// TwinCAT 3 PLC project Intersection
// ProgramVersion: 3.1.4022.2
// libraries:
//   Tc2_Math, * (Beckhoff Automation GmbH)
//   Tc2_Standard, * (Beckhoff Automation GmbH)
//   Tc2_System, * (Beckhoff Automation GmbH)
//   Tc3_Module, * (Beckhoff Automation GmbH)
//   VisuDialogs, * (System)
//   VisuSymbols,3.5.10.0,System
// project tree:
//   01_NorthLight/ NorthLight_Control.TcPOU
//   02_SouthLight/ SouthLight_Control.TcPOU
//   03_EastLight/ EastLight_Control.TcPOU
//   04_WestLight/ WestLight_Control.TcPOU
//   Error Checking/ errorChecking.TcPOU, crosswalkErrorChecks.TcPOU, errorShutdown.TcPOU, lightComboErrorChecks.TcPOU
//   / Glbl.TcGVL, GlobalTextList.TcGTLO, IntersectionVisual.TcVIS, MAIN.TcPOU, PlcTask.TcTTO, Visualization Manager.TcVMO (not stored)
//   Helper Functions/ counterMaintenance.TcPOU, maximum.TcPOU, randomSensors.TcPOU
// real-time tasks:
//   TASK PlcTask: cycle T#1000ms, priority 20, ADS port 350

CONFIGURATION Intersection
    RESOURCE PLC ON TwinCAT3
        TASK PlcTask(INTERVAL := T#1000ms, PRIORITY := 20);
        PROGRAM MAIN WITH PlcTask : MAIN;
    END_RESOURCE
END_CONFIGURATION

// ---- Glbl.TcGVL
{attribute 'qualified_only'}
VAR_GLOBAL
	
	//These track if the lights are on (green/yellow) and are updated in the individual POUs
	northStraightActive : BOOL := FALSE;
	northLeftActive     : BOOL := FALSE;
	southStraightActive : BOOL := FALSE;
	southLeftActive     : BOOL := FALSE;
	eastStraightActive  : BOOL := FALSE;
	eastLeftActive      : BOOL := FALSE;
	westStraightActive  : BOOL := FALSE;
	westLeftActive      : BOOL := FALSE;
	
	//These track the 'how long waiting' for each light combo (state)
	state1Counter : DINT := 0; 							//North Straight and South Straight
	state2Counter : DINT := 0; 							//East Straight and West Straight
	state3Counter : DINT := 0; 							//North Left and South Left
	state4Counter : DINT := 0; 							//East Left and West Left
	state5Counter : DINT := 0; 							//North Straight and Left
	state6Counter : DINT := 0; 							//South Straight and Left
	state7Counter : DINT := 0; 							//East Straight and Left
	state8Counter : DINT := 0; 							//West Straight and Left
	
	//Sensors that indicate 'there is a car here'
	northStraightSensor : BOOL := FALSE;
	northLeftSensor     : BOOL := FALSE;
	southStraightSensor : BOOL := FALSE;
	southLeftSensor     : BOOL := FALSE;
	eastStraightSensor  : BOOL := FALSE;
	eastLeftSensor      : BOOL := FALSE;
	westStraightSensor  : BOOL := FALSE;
	westLeftSensor      : BOOL := FALSE;
	
	//Counters that count the number of cars at a sensor
	northStraightSensorCnt : INT := 0;
	northLeftSensorCnt     : INT := 0;
	southStraightSensorCnt : INT := 0;
	southLeftSensorCnt     : INT := 0;
	eastStraightSensorCnt  : INT := 0;
	eastLeftSensorCnt      : INT := 0;
	westStraightSensorCnt  : INT := 0;
	westLeftSensorCnt      : INT := 0;
	
	//If there is an error (as defined in errorChecking()), this will be true
	error : BOOL := FALSE;
	errorMsg : STRING := 'NULL'; //Contains a message about the error, if applicable
	
END_VAR

// ---- MAIN.TcPOU
PROGRAM MAIN
VAR
END_VAR

//If there is no error, run the code
IF Glbl.error = FALSE THEN
	//If all of the lights are currently red, then decide which light to activate based on the state counters as defined in the Glbl varaible list
	IF Glbl.northStraightActive = FALSE AND Glbl.northLeftActive = FALSE AND Glbl.southStraightActive = FALSE AND Glbl.southLeftActive = FALSE AND Glbl.eastStraightActive = FALSE AND Glbl.eastLeftActive = FALSE AND Glbl.westStraightActive = FALSE AND Glbl.westLeftActive = FALSE THEN
		IF Glbl.state1Counter = maximum() THEN //Turn on North and South Straight lights
			Glbl.northStraightActive := TRUE;
			Glbl.southStraightActive := TRUE;
			Glbl.state1Counter := 0;
		ELSIF Glbl.state2Counter = maximum() AND (Glbl.westStraightSensor = TRUE OR Glbl.eastStraightSensor = TRUE) THEN //Turn on East and West Straight lights
			Glbl.eastStraightActive := TRUE;
			Glbl.westStraightActive := TRUE;
			Glbl.state2Counter := 0;
		ELSIF Glbl.state3Counter = maximum() AND (Glbl.northLeftSensor = TRUE OR Glbl.southLeftSensor = TRUE) THEN //Turn on North and South left lights
			Glbl.northLeftActive := TRUE;
			Glbl.southLeftActive := TRUE;
			Glbl.state3Counter := 0;
		ELSIF Glbl.state4Counter = maximum() AND (Glbl.westLeftSensor = TRUE OR Glbl.eastLeftSensor = TRUE) THEN //Turn on East and West Left lights
			Glbl.eastLeftActive := TRUE;
			Glbl.westLeftActive := TRUE;
			Glbl.state4Counter := 0;
		ELSIF Glbl.state5Counter = maximum() AND (Glbl.northStraightSensor = TRUE OR Glbl.northLeftSensor = TRUE) THEN //Turn on North Left and Straight lights
			Glbl.northStraightActive := TRUE;
			Glbl.northLeftActive := TRUE;
			Glbl.state5Counter := 0;
		ELSIF Glbl.state6Counter = maximum() AND (Glbl.southStraightSensor = TRUE OR Glbl.southLeftSensor = TRUE) THEN //Turn on South Left and Straight lights
			Glbl.southStraightActive := TRUE;
			Glbl.southLeftActive := TRUE;
			Glbl.state6Counter := 0;
		ELSIF Glbl.state7Counter = maximum() AND (Glbl.eastStraightSensor = TRUE OR Glbl.eastLeftSensor = TRUE) THEN //Turn on East Left and Straight lights
			Glbl.eastStraightActive := TRUE;
			Glbl.eastLeftActive := TRUE;
			Glbl.state7Counter := 0;
		ELSIF Glbl.state8Counter = maximum() AND (Glbl.westStraightSensor = TRUE OR Glbl.westLeftSensor = TRUE) THEN //Turn on West Left and Straight lights
			Glbl.westStraightActive := TRUE;
			Glbl.westLeftActive := TRUE;
			Glbl.state8Counter := 0;
		END_IF
	END_IF
	
	//Sets random sensors off
	randomSensors();
	
	//Maintains the part of the counters that fall through the cracks
	counterMaintenance();
	
	//Call each of the lights POUs
	NorthLight_Control();
	SouthLight_Control();
	EastLight_Control();
	WestLight_Control();
ELSE
	//Run the program to shut down system in event of an error
END_IF

END_PROGRAM

// ---- Helper Functions/maximum.TcPOU
FUNCTION maximum : DINT
VAR_INPUT
END_VAR
VAR
	temp : DINT;
END_VAR

temp := MAX(Glbl.state1Counter, Glbl.state2Counter);
temp := MAX(Glbl.state3Counter, temp);
temp := MAX(Glbl.state4Counter, temp);
temp := MAX(Glbl.state5Counter, temp);
temp := MAX(Glbl.state6Counter, temp);
temp := MAX(Glbl.state7Counter, temp);
temp := MAX(Glbl.state8Counter, temp);
maximum := temp;

END_FUNCTION

// ---- Helper Functions/randomSensors.TcPOU
PROGRAM randomSensors
VAR
	DRAND : DRAND;
	Seed : INT;
	Random : LREAL;
END_VAR

Seed := 57; //Set the seed for the random function to some INT
DRAND.Seed := Seed;
DRAND();
Random := DRAND.Num;


IF Random <= 0.200 THEN //Should average once in every 5 seconds (scan time = 1 second, .20/1 probability, 20%
	IF Random <= 0.025 THEN
		Glbl.northStraightSensor := TRUE;
		Glbl.northStraightSensorCnt := Glbl.northStraightSensorCnt + 1;
	ELSIF Random <= 0.050 THEN
		Glbl.northLeftSensor := TRUE;
		Glbl.northLeftSensorCnt := Glbl.northLeftSensorCnt + 1;
	ELSIF Random <= 0.075 THEN
		Glbl.southStraightSensor := TRUE;
		Glbl.southStraightSensorCnt := Glbl.southStraightSensorCnt + 1;
	ELSIF Random <= 0.100 THEN
		Glbl.southLeftSensor := TRUE;
		Glbl.southLeftSensorCnt := Glbl.southLeftSensorCnt + 1;
	ELSIF Random <= 0.125 THEN
		Glbl.eastStraightSensor := TRUE;
		Glbl.eastStraightSensorCnt := Glbl.eastStraightSensorCnt + 1;
	ELSIF Random <= 0.150 THEN
		Glbl.eastLeftSensor := TRUE;
		Glbl.eastLeftSensorCnt := Glbl.eastLeftSensorCnt + 1;
	ELSIF Random <= 0.175 THEN
		Glbl.westStraightSensor := TRUE;
		Glbl.westStraightSensorCnt := Glbl.westStraightSensorCnt + 1;
	ELSE
		Glbl.westLeftSensor := TRUE;
		Glbl.westLeftSensorCnt := Glbl.westLeftSensorCnt + 1;
	END_IF
END_IF

END_PROGRAM

// ---- Helper Functions/counterMaintenance.TcPOU
PROGRAM counterMaintenance
VAR
END_VAR

//Checks all of the sensors and resets the counter appropriatley as a maintenance check

IF Glbl.northStraightSensor = FALSE AND Glbl.southStraightSensor = FALSE THEN
	Glbl.state1Counter := 0;
	Glbl.northStraightSensorCnt := 0;
	Glbl.southStraightSensorCnt := 0;
END_IF

IF Glbl.eastStraightSensor = FALSE AND Glbl.westStraightSensor = FALSE THEN
	Glbl.state2Counter := 0;
	Glbl.eastStraightSensorCnt := 0;
	Glbl.westStraightSensorCnt := 0;
END_IF

IF Glbl.northLeftSensor = FALSE AND Glbl.southLeftSensor = FALSE THEN
	Glbl.state3Counter := 0;
	Glbl.northLeftSensorCnt := 0;
	Glbl.southLeftSensorCnt := 0;
END_IF

IF Glbl.eastLeftSensor = FALSE AND Glbl.westLeftSensor = FALSE THEN
	Glbl.state4Counter := 0;
	Glbl.eastLeftSensorCnt := 0;
	Glbl.westLeftSensorCnt := 0;
END_IF

IF Glbl.northStraightSensor = FALSE AND Glbl.northLeftSensor = FALSE THEN
	Glbl.state5Counter := 0;
	Glbl.northStraightSensorCnt := 0;
	Glbl.northLeftSensorCnt := 0;
END_IF

IF Glbl.southStraightSensor = FALSE AND Glbl.southLeftSensor = FALSE THEN
	Glbl.state6Counter := 0;
	Glbl.southStraightSensorCnt := 0;
	Glbl.southLeftSensorCnt := 0;
END_IF

IF Glbl.eastStraightSensor = FALSE AND Glbl.eastLeftSensor = FALSE THEN
	Glbl.state7Counter := 0;
	Glbl.eastStraightSensorCnt := 0;
	Glbl.eastLeftSensorCnt := 0;
END_IF

IF Glbl.westStraightSensor = FALSE AND Glbl.westLeftSensor = FALSE THEN
	Glbl.state8Counter := 0;
	Glbl.westStraightSensorCnt := 0;
	Glbl.westLeftSensorCnt := 0;
END_IF

END_PROGRAM

// ---- 01_NorthLight/NorthLight_Control.TcPOU
PROGRAM NorthLight_Control
VAR
	StraightGreenLight  : BOOL := FALSE;	//Controls if the green light is on
	StraightYellowLight : BOOL := FALSE;	//Controls if the yellow light is on
	StraightRedLight    : BOOL := TRUE; 	//Controls if the red light is on
	
	StraightOnTimer : INT := 0;				//Tracks how long the light has been on
	
	LeftGreenLight  : BOOL := FALSE;		//Controls if the green light is on
	LeftYellowLight : BOOL := FALSE;		//Controls if the yellow light is on
	leftRedLight    : BOOL := TRUE; 		//Controls if the red light is on
	
	LeftOnTimer : INT := 0;					//Tracks how long the light has been on
	
	CrosswalkLight : BOOL := FALSE;			//Controls if the crosswalk light is on (walk=TRUE)
END_VAR

//If all of the sensors and lights are off, default to N/S straight
IF Glbl.northStraightSensor = FALSE AND  Glbl.northLeftSensor = FALSE AND Glbl.southStraightSensor = FALSE AND Glbl.southLeftSensor = FALSE AND Glbl.eastStraightSensor = FALSE AND Glbl.eastLeftSensor = FALSE AND Glbl.westStraightSensor = FALSE AND Glbl.westLeftSensor = FALSE AND  Glbl.northLeftActive = FALSE AND Glbl.southLeftActive = FALSE AND Glbl.eastStraightActive = FALSE AND Glbl.eastLeftActive = FALSE AND Glbl.westStraightActive = FALSE AND Glbl.westLeftActive = FALSE THEN
	Glbl.northStraightActive := TRUE;
	StraightRedLight := FALSE;
	StraightGreenLight := TRUE;
	
	//Reset the counters, just as a precaution
	Glbl.state1Counter := 0;
	Glbl.state2Counter := 0;
	Glbl.state3Counter := 0;
	Glbl.state4Counter := 0;
	Glbl.state5Counter := 0;
	Glbl.state6Counter := 0;
	Glbl.state7Counter := 0;
	Glbl.state8Counter := 0;
	
ELSE//Control for the straight light if active
	IF Glbl.northStraightActive = TRUE THEN													//If the straight light is set to be active
		IF StraightOnTimer = 0 THEN															//Take off half of the state counter when the light is activated
			Glbl.state1Counter := Glbl.state1Counter - (Glbl.state1Counter/2);
			Glbl.state5Counter := Glbl.state5Counter - (Glbl.state5Counter/2);		
		END_IF
		IF StraightOnTimer <= 10 THEN														//If the light has been on for 10 seconds or less, make it green
			StraightGreenLight := TRUE;
			StraightYellowLight := FALSE;
			StraightRedLight := FALSE;
			StraightOnTimer := StraightOnTimer + 1;											//Incriment the amount of time it has been on by 1
			Glbl.northStraightSensor := FALSE;												//Set the sensor to false
			Glbl.northStraightSensorCnt := MAX(Glbl.northStraightSensorCnt-1, 0);			//Set the car counter to 0
		ELSIF StraightOnTimer <= 13 THEN													//If the light has been on for 11-13 seconds, make it yellow
			StraightGreenLight := FALSE;
			StraightYellowLight := TRUE;
			StraightRedLight := FALSE;
			StraightOnTimer := StraightOnTimer + 1;											//Incriment the amount of time it has been on by 1
		ELSE																				//Once it is done, turn it to red and set it as inactive, reset timer to 0
			StraightGreenLight := FALSE;
			StraightYellowLight := FALSE;
			StraightRedLight := TRUE;
			Glbl.northStraightActive := FALSE;
			StraightOnTimer := 0;	
		END_IF
	END_IF
END_IF

//Control for the left light if active
IF Glbl.northLeftActive = TRUE THEN															//If the left light is set to be active
	IF LeftOnTimer = 0 THEN																	//Take off half of the state counter when the light is activated
		Glbl.state3Counter := Glbl.state3Counter - (Glbl.state3Counter/2);
		Glbl.state5Counter := Glbl.state5Counter - (Glbl.state5Counter/2);	
	END_IF
	IF LeftOnTimer <= 10 THEN																//If the light has been on for 10 seconds or less, make it green
		LeftGreenLight := TRUE;
		LeftYellowLight := FALSE;
		LeftRedLight := FALSE;
		LeftOnTimer := LeftOnTimer + 1;														//Incriment the amount of time it has been on by 1
		Glbl.northLeftSensor := FALSE; 														//Set the sensor to false
		Glbl.northLeftSensorCnt := MAX(Glbl.northLeftSensorCnt-1, 0);
	ELSIF LeftOnTimer <= 13 THEN															//If the light has been on for 11-13 seconds, make it yellow
		LeftGreenLight := FALSE;
		LeftYellowLight := TRUE;
		LeftRedLight := FALSE;
		LeftOnTimer := LeftOnTimer + 1;														//Incriment the amount of time it has been on by 1
	ELSE																					//Once it is done, turn it to red and set it as inactive, reset timer to 0
		LeftGreenLight := FALSE;
		LeftYellowLight := FALSE;
		LeftRedLight := TRUE;
		Glbl.northLeftActive := FALSE;
		LeftOnTimer := 0;	
	END_IF
END_IF

//If the sensor is on and the light is off, incirment the waiting counters
IF Glbl.northStraightSensor = TRUE AND Glbl.northStraightActive = FALSE THEN				//Incriment the striaght counter
	Glbl.state1Counter := Glbl.state1Counter + Glbl.northStraightSensorCnt;
	Glbl.state5Counter := Glbl.state5Counter + Glbl.northStraightSensorCnt;
END_IF
IF Glbl.northLeftSensor = TRUE AND Glbl.northLeftActive = FALSE THEN						//Incriment the left counter
	Glbl.state3Counter := Glbl.state3Counter + Glbl.northLeftSensorCnt;
	Glbl.state5Counter := Glbl.state5Counter + Glbl.northLeftSensorCnt;
END_IF

//Check to see if the crosswalk can be turned on based on the states of the other lights
IF (Glbl.eastStraightActive = TRUE AND Glbl.westStraightActive = TRUE) OR (Glbl.eastStraightActive = TRUE AND Glbl.eastLeftActive = TRUE) THEN
	CrosswalkLight := TRUE;
ELSE
	CrosswalkLight := FALSE;
END_IF

END_PROGRAM

// ---- 02_SouthLight/SouthLight_Control.TcPOU
PROGRAM SouthLight_Control
VAR
	StraightGreenLight  : BOOL := FALSE;	//Controls if the green light is on
	StraightYellowLight : BOOL := FALSE;	//Controls if the yellow light is on
	StraightRedLight    : BOOL := TRUE; 	//Controls if the red light is on
	
	StraightOnTimer : INT := 0;				//Tracks how long the light has been on
	
	LeftGreenLight  : BOOL := FALSE;		//Controls if the green light is on
	LeftYellowLight : BOOL := FALSE;		//Controls if the yellow light is on
	leftRedLight    : BOOL := TRUE; 		//Controls if the red light is on
	
	LeftOnTimer : INT := 0;					//Tracks how long the light has been on
	
	CrosswalkLight : BOOL := FALSE;			//Controls if the crosswalk light is on (walk=TRUE)
END_VAR

//If all of the sensors and lights are off, default to N/S straight
IF Glbl.northStraightSensor = FALSE AND  Glbl.northLeftSensor = FALSE AND Glbl.southStraightSensor = FALSE AND Glbl.southLeftSensor = FALSE AND Glbl.eastStraightSensor = FALSE AND Glbl.eastLeftSensor = FALSE AND Glbl.westStraightSensor = FALSE AND Glbl.westLeftSensor = FALSE AND  Glbl.northLeftActive = FALSE AND Glbl.southLeftActive = FALSE AND Glbl.eastStraightActive = FALSE AND Glbl.eastLeftActive = FALSE AND Glbl.westStraightActive = FALSE AND Glbl.westLeftActive = FALSE THEN
	Glbl.southStraightActive := TRUE;
	StraightRedLight := FALSE;
	StraightGreenLight := TRUE;
ELSE //Control for the straight light if active
IF Glbl.southStraightActive = TRUE THEN														//If the straight light is set to be active
		IF StraightOnTimer = 0 THEN															//Take off half of the state counter when the light is activated
			Glbl.state1Counter := Glbl.state1Counter - (Glbl.state1Counter/2);
			Glbl.state6Counter := Glbl.state6Counter - (Glbl.state6Counter/2);		
		END_IF
		IF StraightOnTimer <= 10 THEN														//If the light has been on for 10 seconds or less, make it green
			StraightGreenLight := TRUE;
			StraightYellowLight := FALSE;
			StraightRedLight := FALSE;
			StraightOnTimer := StraightOnTimer + 1;											//Incriment the amount of time it has been on by 1
			Glbl.southStraightSensor := FALSE;												//Set the sensor to false
			Glbl.southStraightSensorCnt := MAX(Glbl.southStraightSensorCnt-1, 0);			//Set the car counter to 0
		ELSIF StraightOnTimer <= 13 THEN													//If the light has been on for 11-13 seconds, make it yellow
			StraightGreenLight := FALSE;
			StraightYellowLight := TRUE;
			StraightRedLight := FALSE;
			StraightOnTimer := StraightOnTimer + 1;											//Incriment the amount of time it has been on by 1
		ELSE																				//Once it is done, turn it to red and set it as inactive, reset timer to 0
			StraightGreenLight := FALSE;
			StraightYellowLight := FALSE;
			StraightRedLight := TRUE;
			Glbl.southStraightActive := FALSE;
			StraightOnTimer := 0;	
		END_IF
	END_IF
END_IF

//Control for the left light if active
IF Glbl.southLeftActive = TRUE THEN															//If the left light is set to be active
	IF LeftOnTimer = 0 THEN																	//Take off half of the state counter when the light is activated
		Glbl.state3Counter := Glbl.state3Counter - (Glbl.state3Counter/2);
		Glbl.state6Counter := Glbl.state6Counter - (Glbl.state6Counter/2);	
	END_IF
	IF LeftOnTimer <= 10 THEN																//If the light has been on for 10 seconds or less, make it green
		LeftGreenLight := TRUE;
		LeftYellowLight := FALSE;
		LeftRedLight := FALSE;
		LeftOnTimer := LeftOnTimer + 1;														//Incriment the amount of time it has been on by 1
		Glbl.southLeftSensor := FALSE; 														//Set the sensor to false
		Glbl.southLeftSensorCnt := MAX(Glbl.southLeftSensorCnt-1, 0);						//Set the car counter to 0
	ELSIF LeftOnTimer <= 13 THEN															//If the light has been on for 11-13 seconds, make it yellow
		LeftGreenLight := FALSE;
		LeftYellowLight := TRUE;
		LeftRedLight := FALSE;
		LeftOnTimer := LeftOnTimer + 1;														//Incriment the amount of time it has been on by 1
	ELSE																					//Once it is done, turn it to red and set it as inactive, reset timer to 0
		LeftGreenLight := FALSE;
		LeftYellowLight := FALSE;
		LeftRedLight := TRUE;
		Glbl.southLeftActive := FALSE;
		LeftOnTimer := 0;	
	END_IF
END_IF

//If the sensor is on and the light is off, incirment the waiting counters
IF Glbl.southStraightSensor = TRUE AND Glbl.southStraightActive = FALSE THEN				//Incriment the striaght counter
	Glbl.state1Counter := Glbl.state1Counter + Glbl.southStraightSensorCnt;
	Glbl.state6Counter := Glbl.state6Counter + Glbl.southStraightSensorCnt;
END_IF
IF Glbl.southLeftSensor = TRUE AND Glbl.southLeftActive = FALSE THEN						//Incriment the left counter
	Glbl.state3Counter := Glbl.state3Counter + Glbl.southLeftSensorCnt;
	Glbl.state6Counter := Glbl.state6Counter + Glbl.southLeftSensorCnt;
END_IF

//Check to see if the crosswalk can be turned on based on the states of the other lights
IF (Glbl.eastStraightActive = TRUE AND Glbl.westStraightActive = TRUE) OR (Glbl.westStraightActive = TRUE AND Glbl.westLeftActive = TRUE) THEN
	CrosswalkLight := TRUE;
ELSE
	CrosswalkLight := FALSE;
END_IF

END_PROGRAM

// ---- 03_EastLight/EastLight_Control.TcPOU
PROGRAM EastLight_Control
VAR
	StraightGreenLight  : BOOL := FALSE;	//Controls if the green light is on
	StraightYellowLight : BOOL := FALSE;	//Controls if the yellow light is on
	StraightRedLight    : BOOL := TRUE; 	//Controls if the red light is on
	
	StraightOnTimer : INT := 0;				//Tracks how long the light has been on
	
	LeftGreenLight  : BOOL := FALSE;		//Controls if the green light is on
	LeftYellowLight : BOOL := FALSE;		//Controls if the yellow light is on
	leftRedLight    : BOOL := TRUE; 		//Controls if the red light is on
	
	LeftOnTimer : INT := 0;					//Tracks how long the light has been on
	
	CrosswalkLight : BOOL := FALSE;			//Controls if the crosswalk light is on (walk=TRUE)
END_VAR

//Control for the straight light if active
IF Glbl.eastStraightActive = TRUE THEN												//If the straight light is set to be active
	IF StraightOnTimer = 0 THEN														//Take off half of the state counter when the light is activated
		Glbl.state2Counter := Glbl.state2Counter - (Glbl.state2Counter/2);
		Glbl.state7Counter := Glbl.state7Counter - (Glbl.state7Counter/2);		
	END_IF
	IF StraightOnTimer <= 10 THEN													//If the light has been on for 10 seconds or less, make it green
		StraightGreenLight := TRUE;
		StraightYellowLight := FALSE;
		StraightRedLight := FALSE;
		StraightOnTimer := StraightOnTimer + 1;										//Incriment the amount of time it has been on by 1
		Glbl.eastStraightSensor := FALSE;											//Set the sensor to false
		Glbl.eastStraightSensorCnt := MAX(Glbl.eastStraightSensorCnt-1,0);			//Set the car counter to 0
	ELSIF StraightOnTimer <= 13 THEN												//If the light has been on for 11-13 seconds, make it yellow
		StraightGreenLight := FALSE;
		StraightYellowLight := TRUE;
		StraightRedLight := FALSE;
		StraightOnTimer := StraightOnTimer + 1;										//Incriment the amount of time it has been on by 1
	ELSE																			//Once it is done, turn it to red and set it as inactive, reset timer to 0
		StraightGreenLight := FALSE;
		StraightYellowLight := FALSE;
		StraightRedLight := TRUE;
		Glbl.eastStraightActive := FALSE;
		StraightOnTimer := 0;	
	END_IF
END_IF

//Control for the left light if active
IF Glbl.eastLeftActive = TRUE THEN													//If the left light is set to be active
	IF LeftOnTimer = 0 THEN															//Take off half of the state counter when the light is activated
		Glbl.state4Counter := Glbl.state4Counter - (Glbl.state4Counter/2);
		Glbl.state7Counter := Glbl.state7Counter - (Glbl.state7Counter/2);	
	END_IF
	IF LeftOnTimer <= 10 THEN														//If the light has been on for 10 seconds or less, make it green
		LeftGreenLight := TRUE;
		LeftYellowLight := FALSE;
		LeftRedLight := FALSE;
		LeftOnTimer := LeftOnTimer + 1;												//Incriment the amount of time it has been on by 1
		Glbl.eastLeftSensor := FALSE; 												//Set the sensor to false
		Glbl.eastLeftSensorCnt := MAX(Glbl.eastLeftSensorCnt-1,0);					//Set the car counter to 0
	ELSIF LeftOnTimer <= 13 THEN													//If the light has been on for 11-13 seconds, make it yellow
		LeftGreenLight := FALSE;
		LeftYellowLight := TRUE;
		LeftRedLight := FALSE;
		LeftOnTimer := LeftOnTimer + 1;												//Incriment the amount of time it has been on by 1
	ELSE																			//Once it is done, turn it to red and set it as inactive, reset timer to 0
		LeftGreenLight := FALSE;
		LeftYellowLight := FALSE;
		LeftRedLight := TRUE;
		Glbl.eastLeftActive := FALSE;
		LeftOnTimer := 0;	
	END_IF
END_IF

//If the sensor is on and the light is off, incirment the waiting counters
IF Glbl.eastStraightSensor = TRUE AND Glbl.eastStraightActive = FALSE THEN			//Incriment the striaght counter
	Glbl.state2Counter := Glbl.state2Counter + Glbl.eastStraightSensorCnt;
	Glbl.state7Counter := Glbl.state7Counter + Glbl.eastStraightSensorCnt;
END_IF
IF Glbl.eastLeftSensor = TRUE AND Glbl.eastLeftActive = FALSE THEN					//Incriment the left counter
	Glbl.state4Counter := Glbl.state4Counter + Glbl.eastLeftSensorCnt;
	Glbl.state7Counter := Glbl.state7Counter + Glbl.eastLeftSensorCnt;
END_IF

//Check to see if the crosswalk can be turned on based on the states of the other lights
IF (Glbl.northStraightActive = TRUE AND Glbl.southStraightActive = TRUE) OR (Glbl.southStraightActive = TRUE AND Glbl.southLeftActive = TRUE) THEN
	CrosswalkLight := TRUE;
ELSE
	CrosswalkLight := FALSE;
END_IF

END_PROGRAM

// ---- 04_WestLight/WestLight_Control.TcPOU
PROGRAM WestLight_Control
VAR
	StraightGreenLight  : BOOL := FALSE;	//Controls if the green light is on
	StraightYellowLight : BOOL := FALSE;	//Controls if the yellow light is on
	StraightRedLight    : BOOL := TRUE; 	//Controls if the red light is on
	
	StraightOnTimer : INT := 0;				//Tracks how long the light has been on
	
	LeftGreenLight  : BOOL := FALSE;		//Controls if the green light is on
	LeftYellowLight : BOOL := FALSE;		//Controls if the yellow light is on
	leftRedLight    : BOOL := TRUE; 		//Controls if the red light is on
	
	LeftOnTimer : INT := 0;					//Tracks how long the light has been on
	
	CrosswalkLight : BOOL := FALSE;			//Controls if the crosswalk light is on (walk=TRUE)
END_VAR

//Control for the straight light if active
IF Glbl.westStraightActive = TRUE THEN													//If the straight light is set to be active
	IF StraightOnTimer = 0 THEN															//Take off half of the state counter when the light is activated
		Glbl.state2Counter := Glbl.state2Counter - (Glbl.state2Counter/2);
		Glbl.state8Counter := Glbl.state8Counter - (Glbl.state8Counter/2);		
	END_IF
	IF StraightOnTimer <= 10 THEN														//If the light has been on for 10 seconds or less, make it green
		StraightGreenLight := TRUE;
		StraightYellowLight := FALSE;
		StraightRedLight := FALSE;
		StraightOnTimer := StraightOnTimer + 1;											//Incriment the amount of time it has been on by 1
		Glbl.westStraightSensor := FALSE;												//Set the sensor to false
		Glbl.westStraightSensorCnt := MAX(Glbl.westStraightSensorCnt-1,0);				//Set the car counter to 0
	ELSIF StraightOnTimer <= 13 THEN													//If the light has been on for 11-13 seconds, make it yellow
		StraightGreenLight := FALSE;
		StraightYellowLight := TRUE;
		StraightRedLight := FALSE;
		StraightOnTimer := StraightOnTimer + 1;											//Incriment the amount of time it has been on by 1
	ELSE																				//Once it is done, turn it to red and set it as inactive, reset timer to 0
		StraightGreenLight := FALSE;
		StraightYellowLight := FALSE;
		StraightRedLight := TRUE;
		Glbl.westStraightActive := FALSE;
		StraightOnTimer := 0;	
	END_IF
END_IF

//Control for the left light if active
IF Glbl.westLeftActive = TRUE THEN														//If the left light is set to be active
	IF LeftOnTimer = 0 THEN																//Take off half of the state counter when the light is activated
		Glbl.state4Counter := Glbl.state4Counter - (Glbl.state4Counter/2);
		Glbl.state8Counter := Glbl.state8Counter - (Glbl.state8Counter/2);	
	END_IF
	IF LeftOnTimer <= 10 THEN															//If the light has been on for 10 seconds or less, make it green
		LeftGreenLight := TRUE;
		LeftYellowLight := FALSE;
		LeftRedLight := FALSE;
		LeftOnTimer := LeftOnTimer + 1;													//Incriment the amount of time it has been on by 1
		Glbl.westLeftSensor := FALSE; 													//Set the sensor to false
		Glbl.westLeftSensorCnt := MAX(Glbl.westLeftSensorCnt-1,0);						//Set the car counter to 0
	ELSIF LeftOnTimer <= 13 THEN														//If the light has been on for 11-13 seconds, make it yellow
		LeftGreenLight := FALSE;
		LeftYellowLight := TRUE;
		LeftRedLight := FALSE;
		LeftOnTimer := LeftOnTimer + 1;													//Incriment the amount of time it has been on by 1
	ELSE																				//Once it is done, turn it to red and set it as inactive, reset timer to 0
		LeftGreenLight := FALSE;
		LeftYellowLight := FALSE;
		LeftRedLight := TRUE;
		Glbl.westLeftActive := FALSE;
		LeftOnTimer := 0;	
	END_IF
END_IF

//If the sensor is on and the light is off, incirment the waiting counters
IF Glbl.westStraightSensor = TRUE AND Glbl.westStraightActive = FALSE THEN
	Glbl.state2Counter := Glbl.state2Counter + Glbl.westStraightSensorCnt;
	Glbl.state8Counter := Glbl.state8Counter + Glbl.westStraightSensorCnt;
END_IF
IF Glbl.westLeftSensor = TRUE AND Glbl.westLeftActive = FALSE THEN
	Glbl.state4Counter := Glbl.state4Counter + Glbl.westLeftSensorCnt;
	Glbl.state8Counter := Glbl.state8Counter + Glbl.westLeftSensorCnt;
END_IF

//Check to see if the crosswalk can be turned on based on the states of the other lights
IF (Glbl.northStraightActive = TRUE AND Glbl.southStraightActive = TRUE) OR (Glbl.northStraightActive = TRUE AND Glbl.northLeftActive = TRUE) THEN
	CrosswalkLight := TRUE;
ELSE
	CrosswalkLight := FALSE;
END_IF

END_PROGRAM

// ---- Error Checking/errorChecking.TcPOU
PROGRAM errorChecking
VAR
END_VAR

//If there are more than two lights active at any time
IF (BOOL_TO_INT(Glbl.northStraightActive) + BOOL_TO_INT(Glbl.northLeftActive) + BOOL_TO_INT(Glbl.southStraightActive) + BOOL_TO_INT(Glbl.southLeftActive) + BOOL_TO_INT(Glbl.eastStraightActive) + BOOL_TO_INT(Glbl.eastLeftActive) + BOOL_TO_INT(Glbl.westStraightActive) + BOOL_TO_INT(Glbl.westLeftActive)) > 2 THEN
	Glbl.error := TRUE;
	Glbl.errorMsg := 'Too many lights active';
END_IF

//Checks to make sure that there are no lights that would interfere with a crosswalk being on
crosswalkErrorChecks();

//Checks to make sure that there are no lights that would interfere with another light being on
lightComboErrorChecks();

END_PROGRAM

// ---- Error Checking/crosswalkErrorChecks.TcPOU
PROGRAM crosswalkErrorChecks
VAR
END_VAR
VAR // added by the converter: edge detectors and wires of the graphical bodies
    _w1, _w2, _w3, _w4 : BOOL;
END_VAR

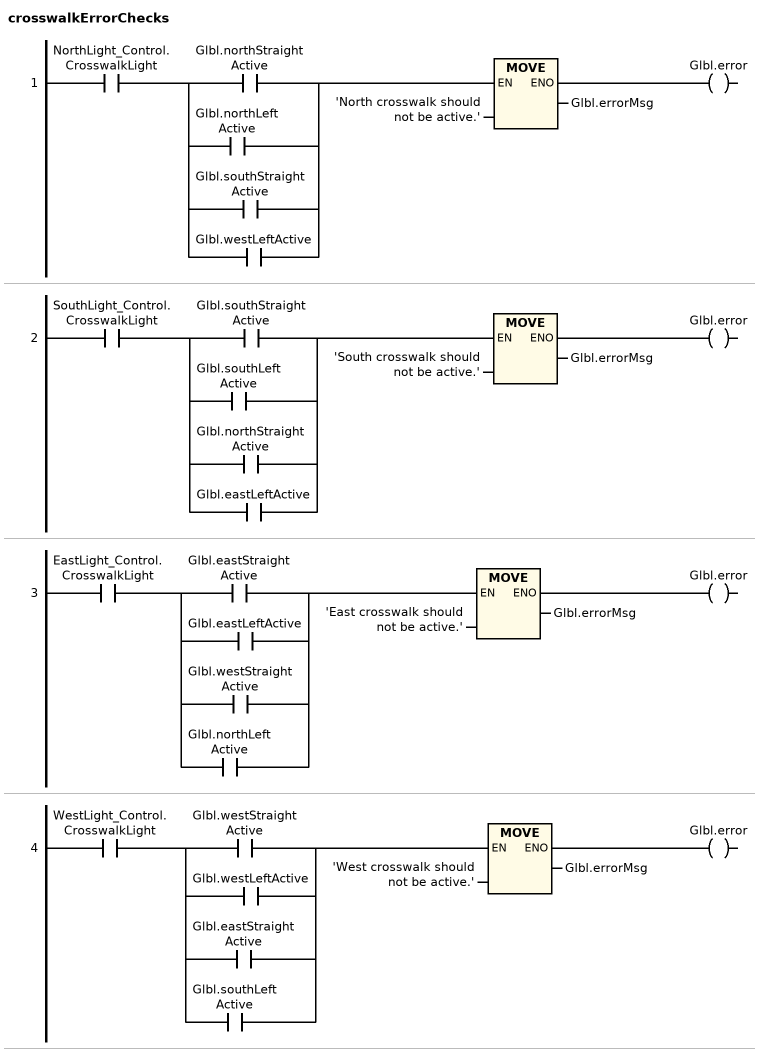
// NETWORK 1
_w1 := NorthLight_Control.CrosswalkLight AND (Glbl.northStraightActive OR Glbl.northLeftActive OR Glbl.southStraightActive OR Glbl.westLeftActive);
IF _w1 THEN Glbl.errorMsg := 'North crosswalk should not be active.'; END_IF
Glbl.error := _w1;

// NETWORK 2
_w2 := SouthLight_Control.CrosswalkLight AND (Glbl.southStraightActive OR Glbl.southLeftActive OR Glbl.northStraightActive OR Glbl.eastLeftActive);
IF _w2 THEN Glbl.errorMsg := 'South crosswalk should not be active.'; END_IF
Glbl.error := _w2;

// NETWORK 3
_w3 := EastLight_Control.CrosswalkLight AND (Glbl.eastStraightActive OR Glbl.eastLeftActive OR Glbl.westStraightActive OR Glbl.northLeftActive);
IF _w3 THEN Glbl.errorMsg := 'East crosswalk should not be active.'; END_IF
Glbl.error := _w3;

// NETWORK 4
_w4 := WestLight_Control.CrosswalkLight AND (Glbl.westStraightActive OR Glbl.westLeftActive OR Glbl.eastStraightActive OR Glbl.southLeftActive);
IF _w4 THEN Glbl.errorMsg := 'West crosswalk should not be active.'; END_IF
Glbl.error := _w4;

END_PROGRAM

// ---- Error Checking/lightComboErrorChecks.TcPOU
PROGRAM lightComboErrorChecks
VAR
END_VAR
VAR // added by the converter: edge detectors and wires of the graphical bodies
    _w1, _w2, _w3, _w4, _w5, _w6, _w7, _w8 : BOOL;
END_VAR

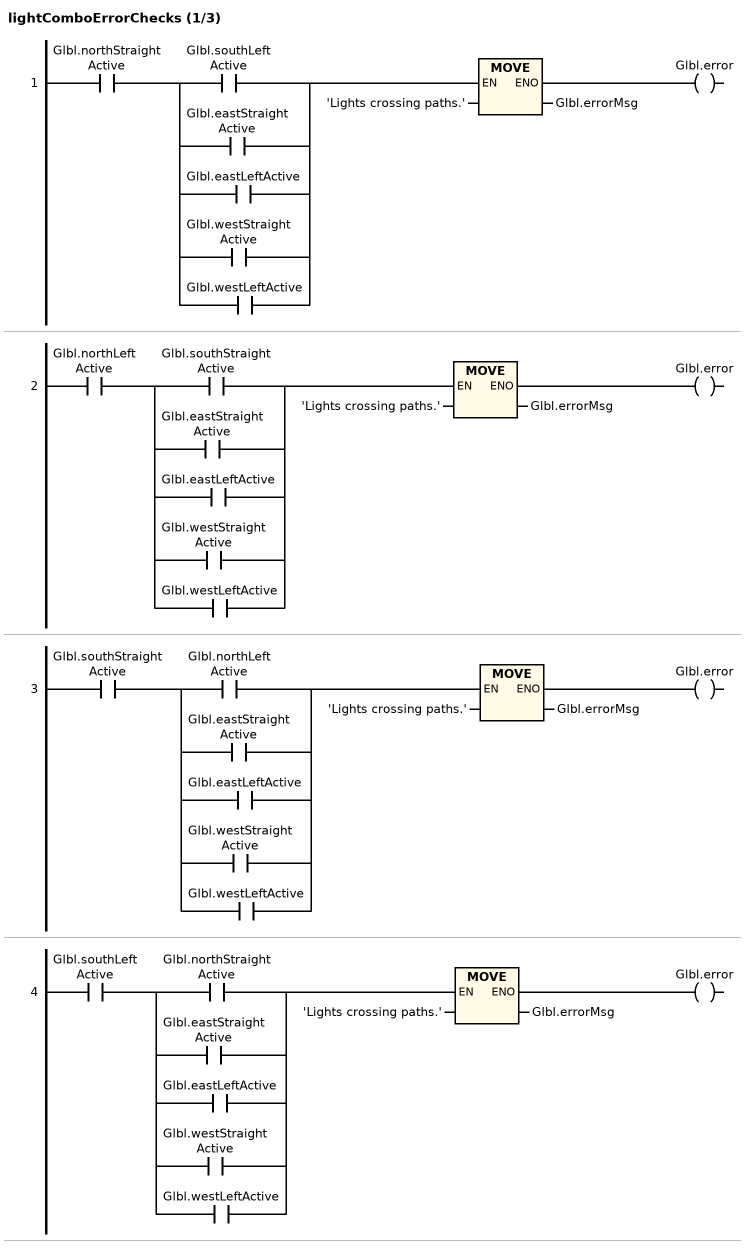
// NETWORK 1
_w1 := Glbl.northStraightActive AND (Glbl.southLeftActive OR Glbl.eastStraightActive OR Glbl.eastLeftActive OR Glbl.westStraightActive OR Glbl.westLeftActive);
IF _w1 THEN Glbl.errorMsg := 'Lights crossing paths.'; END_IF
Glbl.error := _w1;

// NETWORK 2
_w2 := Glbl.northLeftActive AND (Glbl.southStraightActive OR Glbl.eastStraightActive OR Glbl.eastLeftActive OR Glbl.westStraightActive OR Glbl.westLeftActive);
IF _w2 THEN Glbl.errorMsg := 'Lights crossing paths.'; END_IF
Glbl.error := _w2;

// NETWORK 3
_w3 := Glbl.southStraightActive AND (Glbl.northLeftActive OR Glbl.eastStraightActive OR Glbl.eastLeftActive OR Glbl.westStraightActive OR Glbl.westLeftActive);
IF _w3 THEN Glbl.errorMsg := 'Lights crossing paths.'; END_IF
Glbl.error := _w3;

// NETWORK 4
_w4 := Glbl.southLeftActive AND (Glbl.northStraightActive OR Glbl.eastStraightActive OR Glbl.eastLeftActive OR Glbl.westStraightActive OR Glbl.westLeftActive);
IF _w4 THEN Glbl.errorMsg := 'Lights crossing paths.'; END_IF
Glbl.error := _w4;

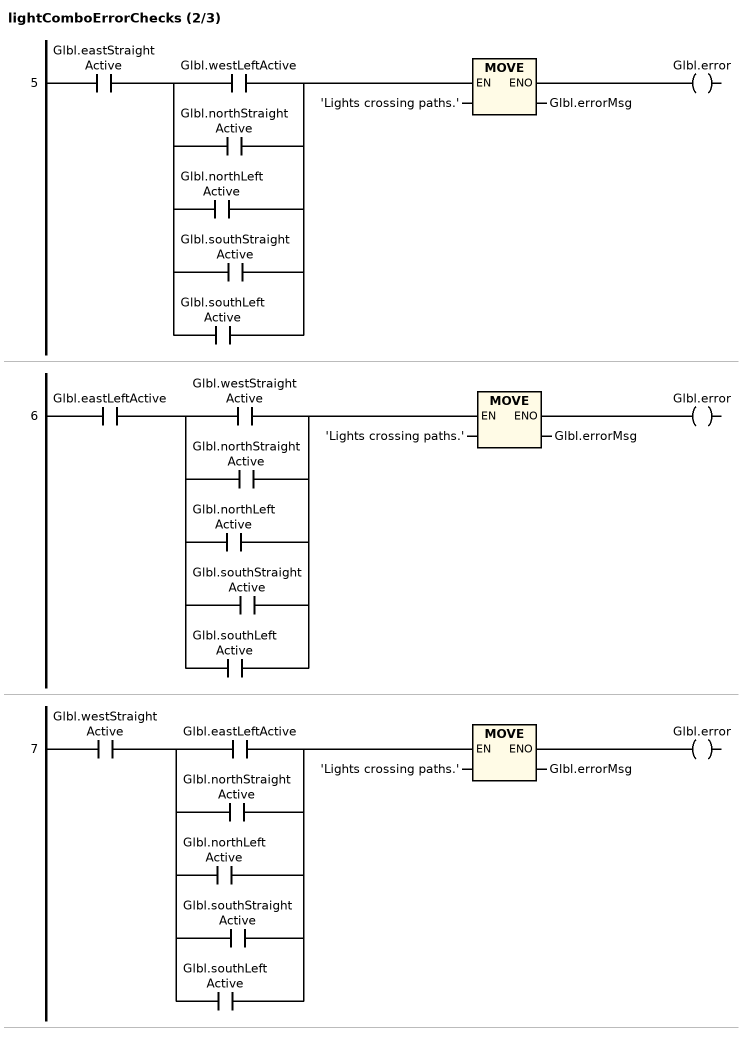
// NETWORK 5
_w5 := Glbl.eastStraightActive AND (Glbl.westLeftActive OR Glbl.northStraightActive OR Glbl.northLeftActive OR Glbl.southStraightActive OR Glbl.southLeftActive);
IF _w5 THEN Glbl.errorMsg := 'Lights crossing paths.'; END_IF
Glbl.error := _w5;

// NETWORK 6
_w6 := Glbl.eastLeftActive AND (Glbl.westStraightActive OR Glbl.northStraightActive OR Glbl.northLeftActive OR Glbl.southStraightActive OR Glbl.southLeftActive);
IF _w6 THEN Glbl.errorMsg := 'Lights crossing paths.'; END_IF
Glbl.error := _w6;

// NETWORK 7
_w7 := Glbl.westStraightActive AND (Glbl.eastLeftActive OR Glbl.northStraightActive OR Glbl.northLeftActive OR Glbl.southStraightActive OR Glbl.southLeftActive);
IF _w7 THEN Glbl.errorMsg := 'Lights crossing paths.'; END_IF
Glbl.error := _w7;

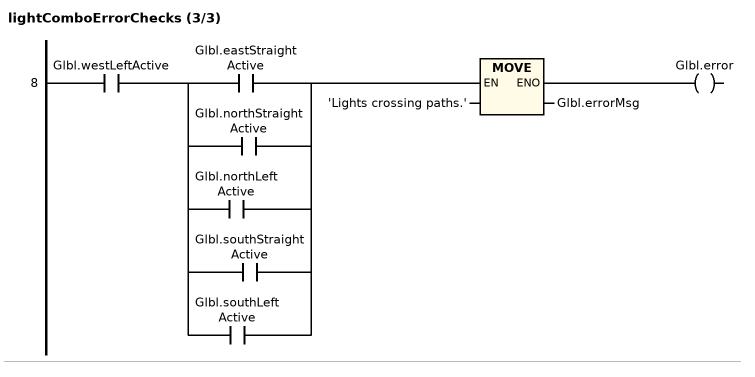
// NETWORK 8
_w8 := Glbl.westLeftActive AND (Glbl.eastStraightActive OR Glbl.northStraightActive OR Glbl.northLeftActive OR Glbl.southStraightActive OR Glbl.southLeftActive);
IF _w8 THEN Glbl.errorMsg := 'Lights crossing paths.'; END_IF
Glbl.error := _w8;

END_PROGRAM

// ---- Error Checking/errorShutdown.TcPOU
PROGRAM errorShutdown
VAR
END_VAR

//Set all of the lights to false
Glbl.northStraightActive := FALSE;
Glbl.northLeftActive := FALSE;
Glbl.southStraightActive := FALSE;
Glbl.southLeftActive := FALSE;
Glbl.eastStraightActive := FALSE;
Glbl.eastLeftActive := FALSE;
Glbl.westStraightActive := FALSE;
Glbl.westLeftActive := FALSE;


//Turn all the lights to red, turn the crosswalks to red, make sure no cars can go until the error is resolved
NorthLight_Control.StraightGreenLight := FALSE;
NorthLight_Control.StraightYellowLight := FALSE;
NorthLight_Control.StraightRedLight := TRUE;
NorthLight_Control.LeftGreenLight := FALSE;
NorthLight_Control.LeftYellowLight := FALSE;
NorthLight_Control.LeftRedLight := TRUE;
NorthLight_Control.CrosswalkLight := FALSE;

SouthLight_Control.StraightGreenLight := FALSE;
SouthLight_Control.StraightYellowLight := FALSE;
SouthLight_Control.StraightRedLight := TRUE;
SouthLight_Control.LeftGreenLight := FALSE;
SouthLight_Control.LeftYellowLight := FALSE;
SouthLight_Control.LeftRedLight := TRUE;
SouthLight_Control.CrosswalkLight := FALSE;

EastLight_Control.StraightGreenLight := FALSE;
EastLight_Control.StraightYellowLight := FALSE;
EastLight_Control.StraightRedLight := TRUE;
EastLight_Control.LeftGreenLight := FALSE;
EastLight_Control.LeftYellowLight := FALSE;
EastLight_Control.LeftRedLight := TRUE;
EastLight_Control.CrosswalkLight := FALSE;

WestLight_Control.StraightGreenLight := FALSE;
WestLight_Control.StraightYellowLight := FALSE;
WestLight_Control.StraightRedLight := TRUE;
WestLight_Control.LeftGreenLight := FALSE;
WestLight_Control.LeftYellowLight := FALSE;
WestLight_Control.LeftRedLight := TRUE;
WestLight_Control.CrosswalkLight := FALSE;

END_PROGRAM

// ---- GlobalTextList.TcGTLO
TEXTLIST GlobalTextList
  463 = '%d'
  761 = '("North/South Straight: %d", glbl.state1counter)'
  528 = 'ALERT'
  359 = 'East'
  684 = 'East Straight/Left:\t%d'
  994 = 'East Straight/Left: %d'
  800 = 'East/West Left:\t\t%d'
  485 = 'East/West Left:\t%d'
  620 = 'East/West Left: %d'
  565 = 'East/West Straight:\t%d'
  679 = 'East/West Straight: %d'
  43 = 'Eat/West Left: %d'
  714 = 'Eat/West Straight: %d'
  263 = 'ERROR'
  808 = 'ERROR $n %s'
  911 = 'ERROR /n %s'
  572 = 'Glbl.state1counter'
  276 = 'Message: %s'
  799 = 'North'
  380 = 'North Straight/Left:\t\t%d'
  259 = 'North Straight/Left:\t%d'
  77 = 'North Straight/Left: %d'
  727 = 'North/South Left:\t%d'
  288 = 'North/South Left: %d'
  280 = 'North/South Straight:\t%d'
  699 = 'North/South Straight: %d'
  614 = 'North/South Straight: %d"'
  840 = 'North?South Left: %d'
  817 = 'Queue East Left'
  877 = 'Queue East Straight'
  226 = 'Queue North Left'
  535 = 'Queue North Straight'
  185 = 'Queue South Left'
  295 = 'Queue South Straight'
  71 = 'Queue West Left'
  564 = 'Queue West Straight'
  586 = 'South'
  794 = 'South Straight/Left: \t%d'
  315 = 'South Straight/Left: %d'
  599 = 'West'
  299 = 'West Straight/Left:\t%d'
END_TEXTLIST

// ---- IntersectionVisual.TcVIS
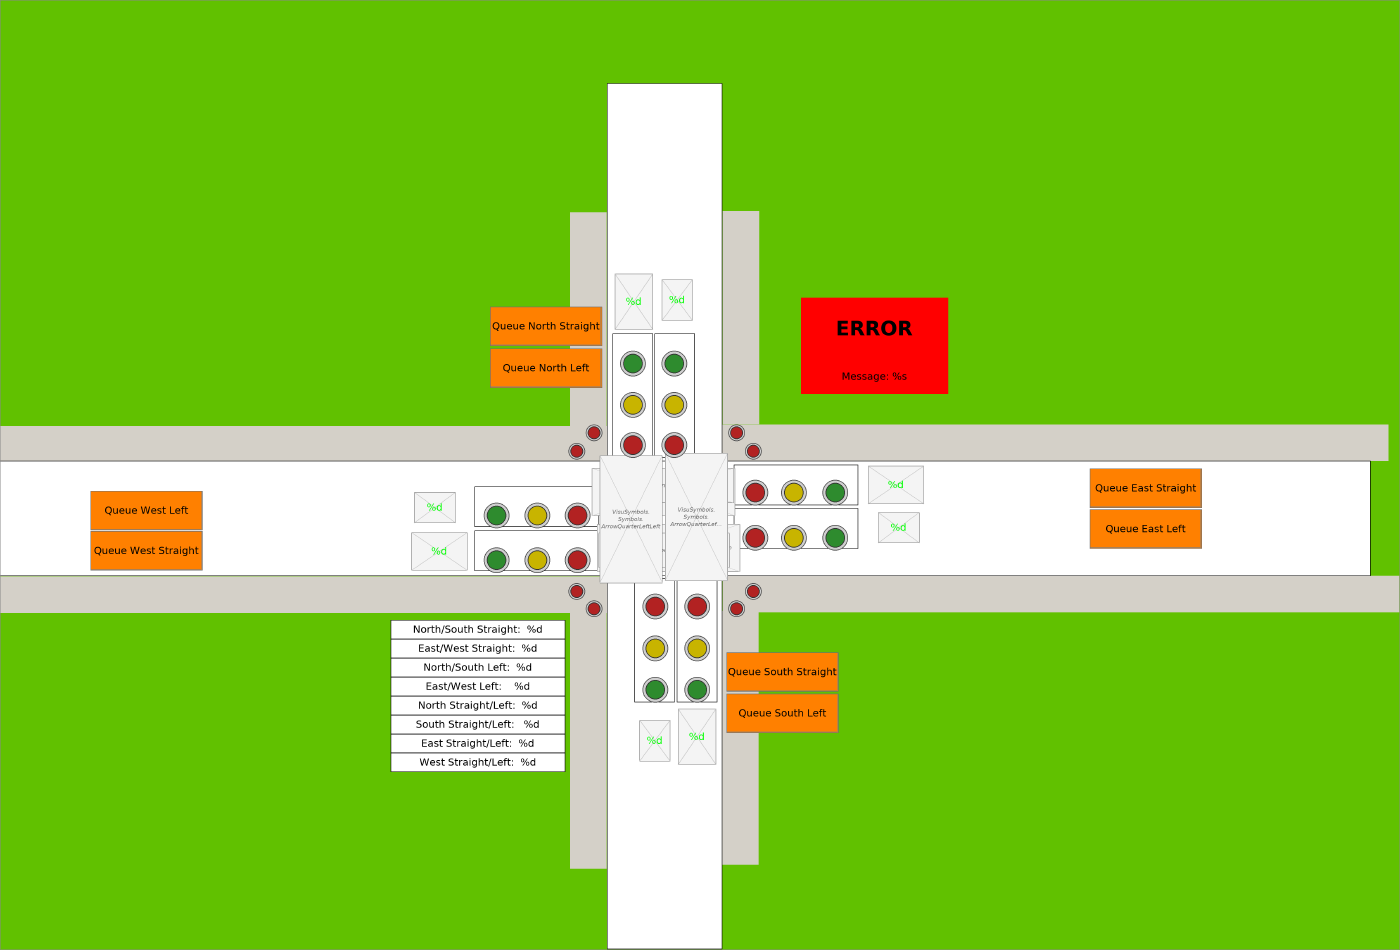
VISUALIZATION IntersectionVisual  // 2505x1701
    Rectangle (1292,1094 65x454)
    Rectangle (1020,1095 65x460)
    Rectangle (1020,380 65x384)
    Rectangle (1293,378 65x381)
    Rectangle (1293,1031 1210x65)
    Rectangle (0,1032 1088x65)
    Rectangle (0,763 1086x65)
    Rectangle (1291,760 1193x65)
    Rectangle (1086,149 206x1550)
    Rectangle (0,825 2452x206)
    Label (2086,901 197x64), "East"
    Label (1090,415 197x64), "North"
    Label (1091,1392 197x64), "South"
    Label (14,891 197x64), "West"
    RoundedRectangle (1313,832 222x72)
    Lamp1 (1394,840 53x84), variable: EastLight_Control.StraightYellowLight, style: Lamp-Lamp1-Yellow
    Lamp1 (1468,840 53x84), variable: EastLight_Control.StraightGreenLight, style: Lamp-Lamp1-Green
    Image (1553,834 100x68), "%d", text variable: Glbl.eastStraightSensorCnt, invisible if: NOT Glbl.eastStraightSensor, image: VisuSymbols.Symbols.ArrowBoldLeft
    RoundedRectangle (1313,910 222x72)
    Lamp1 (1394,921 53x84), variable: EastLight_Control.LeftYellowLight, style: Lamp-Lamp1-Yellow
    Lamp1 (1468,921 53x84), variable: EastLight_Control.LeftGreenLight, style: Lamp-Lamp1-Green
    Image (1571,917 74x55), "%d", text variable: Glbl.eastLeftSensorCnt, colour toggle: Glbl.eastLeftSensor, invisible if: Not Glbl.eastLeftSensor, image: VisuSymbols.Symbols.ArrowBoldDown
    Button (1950,839 200x70), "Queue East Straight"
        OnMouseDown: execute { Glbl.eastStraightSensor := TRUE; Glbl.eastStraightSensorCnt := Glbl.eastStraightSensorCnt + 1; }
    Button (1950,912 200x70), "Queue East Left"
        OnMouseDown: execute { Glbl.eastLeftSensor := TRUE; Glbl.eastLeftSensorCnt := Glbl.eastLeftSensorCnt + 1; }
    RoundedRectangle (849,871 222x72)
    RoundedRectangle (849,950 222x72)
    Lamp1 (1007,881 53x84), variable: WestLight_Control.LeftRedLight, style: Lamp-Lamp1-Red
    Lamp1 (935,881 53x84), variable: WestLight_Control.LeftYellowLight, style: Lamp-Lamp1-Yellow
    Lamp1 (862,881 53x84), variable: WestLight_Control.LeftGreenLight, style: Lamp-Lamp1-Green
    Lamp1 (1007,961 53x84), variable: WestLight_Control.StraightRedLight, style: Lamp-Lamp1-Red
    Lamp1 (935,961 53x84), variable: WestLight_Control.StraightYellowLight, style: Lamp-Lamp1-Yellow
    Lamp1 (862,961 53x84), variable: WestLight_Control.StraightGreenLight, style: Lamp-Lamp1-Green
    Image (736,953 100x68), "%d", text variable: Glbl.westStraightSensorCnt, invisible if: Not Glbl.westStraightSensor, image: VisuSymbols.Symbols.ArrowBoldRight
    Image (741,881 74x55), "%d", text variable: Glbl.westLeftSensorCnt, invisible if: Not Glbl.westLeftSensor, image: VisuSymbols.Symbols.ArrowBoldUp
    Button (162,951 200x70), "Queue West Straight"
        OnMouseDown: execute { Glbl.westStraightSensor := TRUE; Glbl.westStraightSensorCnt := Glbl.westStraightSensorCnt + 1; }
    Button (162,879 200x70), "Queue West Left"
        OnMouseDown: execute { Glbl.westLeftSensor := TRUE; Glbl.westLeftSensorCnt := Glbl.westLeftSensorCnt + 1; }
    Lamp1 (1301,1070 34x40), variable: SouthLight_Control.CrosswalkLight, invisible if: NOT SouthLight_Control.CrosswalkLight, style: Lamp-Lamp1-Green
    Lamp1 (1331,1039 34x40), variable: EastLight_Control.CrosswalkLight, invisible if: NOT EastLight_Control.CrosswalkLight, style: Lamp-Lamp1-Green
    Lamp1 (1046,1070 34x40), variable: SouthLight_Control.CrosswalkLight, invisible if: NOT SouthLight_Control.CrosswalkLight, style: Lamp-Lamp1-Green
    Lamp1 (1015,1039 34x40), variable: WestLight_Control.CrosswalkLight, invisible if: NOT WestLight_Control.CrosswalkLight, style: Lamp-Lamp1-Green
    Lamp1 (1331,788 34x40), variable: EastLight_Control.CrosswalkLight, invisible if: NOT EastLight_Control.CrosswalkLight, style: Lamp-Lamp1-Green
    Lamp1 (1301,755 34x40), variable: NorthLight_Control.CrosswalkLight, invisible if: NOT NorthLight_Control.CrosswalkLight, style: Lamp-Lamp1-Green
    Lamp1 (1015,788 34x40), variable: WestLight_Control.CrosswalkLight, invisible if: NOT WestLight_Control.CrosswalkLight, style: Lamp-Lamp1-Green
    Lamp1 (1046,755 34x40), variable: NorthLight_Control.CrosswalkLight, invisible if: NOT NorthLight_Control.CrosswalkLight, style: Lamp-Lamp1-Green
    Lamp1 (1331,788 34x40), variable: NOT EastLight_Control.CrosswalkLight, invisible if: EastLight_Control.CrosswalkLight, style: Lamp-Lamp1-Red
    Lamp1 (1301,755 34x40), variable: NOT NorthLight_Control.CrosswalkLight, invisible if: NorthLight_Control.CrosswalkLight, style: Lamp-Lamp1-Red
    Lamp1 (1331,1039 34x40), variable: NOT EastLight_Control.CrosswalkLight, invisible if: EastLight_Control.CrosswalkLight, style: Lamp-Lamp1-Red
    Lamp1 (1301,1070 34x40), variable: NOT SouthLight_Control.CrosswalkLight, invisible if: SouthLight_Control.CrosswalkLight, style: Lamp-Lamp1-Red
    Lamp1 (1046,755 34x40), variable: NOT NorthLight_Control.CrosswalkLight, invisible if: NorthLight_Control.CrosswalkLight, style: Lamp-Lamp1-Red
    Lamp1 (1015,788 34x40), variable: NOT WestLight_Control.CrosswalkLight, invisible if: WestLight_Control.CrosswalkLight, style: Lamp-Lamp1-Red
    Lamp1 (1015,1039 34x40), variable: NOT WestLight_Control.CrosswalkLight, invisible if: WestLight_Control.CrosswalkLight, style: Lamp-Lamp1-Red
    Lamp1 (1046,1070 34x40), variable: NOT SouthLight_Control.CrosswalkLight, invisible if: SouthLight_Control.CrosswalkLight, style: Lamp-Lamp1-Red
    Image (1059,838 256x85), invisible if: NOT Glbl.westLeftActive, image: VisuSymbols.Symbols.ArrowQuarterLeftUp
    Image (1068,938 256x85), invisible if: NOT Glbl.eastLeftActive, image: VisuSymbols.Symbols.ArrowQuarterLeftDown
    Image (1079,838 234x62), invisible if: NOT Glbl.eastStraightActive, image: VisuSymbols.Symbols.ArrowBoldLeft
    Image (1071,954 234x62), invisible if: Not Glbl.westStraightActive, image: VisuSymbols.Symbols.ArrowBoldRight
    RoundedRectangle (1211,1035 72x222)
    RoundedRectangle (1135,1035 72x222)
    Lamp1 (1221,1044 53x84), variable: SouthLight_Control.StraightRedLight, style: Lamp-Lamp1-Red
    Lamp1 (1146,1044 53x84), variable: SouthLight_Control.LeftRedLight, style: Lamp-Lamp1-Red
    Lamp1 (1146,1119 53x84), variable: SouthLight_Control.LeftYellowLight, style: Lamp-Lamp1-Yellow
    Lamp1 (1221,1119 53x84), variable: SouthLight_Control.StraightYellowLight, style: Lamp-Lamp1-Yellow
    Lamp1 (1146,1193 53x84), variable: SouthLight_Control.LeftGreenLight, style: Lamp-Lamp1-Green
    Lamp1 (1221,1193 53x84), variable: SouthLight_Control.StraightGreenLight, style: Lamp-Lamp1-Green
    Button (1300,1168 200x70), "Queue South Straight"
        OnMouseDown: execute { Glbl.southStraightSensor := TRUE; Glbl.southStraightSensorCnt := Glbl.southStraightSensorCnt + 1; }
    Button (1300,1242 200x70), "Queue South Left"
        OnMouseDown: execute { Glbl.southLeftSensor := TRUE; Glbl.southLeftSensorCnt := Glbl.southLeftSensorCnt + 1; }
    RoundedRectangle (1096,597 72x222)
    RoundedRectangle (1171,597 72x222)
    Image (1144,1289 55x74), "%d", text variable: Glbl.southLeftSensorCnt, invisible if: NOT Glbl.southLeftSensor, image: VisuSymbols.Symbols.ArrowBoldLeft
    Image (1213,1269 68x100), "%d", text variable: Glbl.southStraightSensorCnt, invisible if: Not Glbl.southStraightSensor, image: VisuSymbols.Symbols.ArrowBoldUp
    Image (1096,822 62x193), colour toggle: Glbl.eastLeftSensor, invisible if: Not Glbl.northStraightActive, image: VisuSymbols.Symbols.ArrowBoldDown
    Image (1215,841 62x193), invisible if: Not Glbl.southStraightActive, image: VisuSymbols.Symbols.ArrowBoldUp
    Image (1190,811 112x229), invisible if: NOT Glbl.northLeftActive, image: VisuSymbols.Symbols.ArrowQuarterLeftRight
    Image (1073,815 112x229), invisible if: NOT Glbl.southLeftActive, image: VisuSymbols.Symbols.ArrowQuarterLeftLeft
    Lamp1 (1106,755 53x84), variable: NorthLight_Control.StraightRedLight, style: Lamp-Lamp1-Red
    Lamp1 (1106,683 53x84), variable: NorthLight_Control.StraightYellowLight, style: Lamp-Lamp1-Yellow
    Lamp1 (1106,609 53x84), variable: NorthLight_Control.StraightGreenLight, style: Lamp-Lamp1-Green
    Lamp1 (1180,755 53x84), variable: NorthLight_Control.LeftRedLight, style: Lamp-Lamp1-Red
    Lamp1 (1180,683 53x84), variable: NorthLight_Control.LeftYellowLight, style: Lamp-Lamp1-Yellow
    Lamp1 (1180,609 53x84), variable: NorthLight_Control.LeftGreenLight, style: Lamp-Lamp1-Green
    Button (877,549 200x70), "Queue North Straight"
        OnMouseDown: execute { Glbl.northStraightSensor := TRUE; Glbl.northStraightSensorCnt := Glbl.northStraightSensorCnt + 1; }
    Button (877,624 200x70), "Queue North Left"
        OnMouseDown: execute { Glbl.northLeftSensor := TRUE; Glbl.northLeftSensorCnt := Glbl.northLeftSensorCnt + 1; }
    Image (1100,490 68x100), "%d", text variable: Glbl.northStraightSensorCnt, colour toggle: Glbl.eastLeftSensor, invisible if: Not Glbl.northStraightSensor, image: VisuSymbols.Symbols.ArrowBoldDown
    Image (1184,500 55x74), "%d", text variable: Glbl.northLeftSensorCnt, invisible if: Not Glbl.northLeftSensor, image: VisuSymbols.Symbols.ArrowBoldRight
    Lamp1 (1325,921 53x84), variable: EastLight_Control.leftRedLight, style: Lamp-Lamp1-Red
    Lamp1 (1325,840 53x84), variable: EastLight_Control.StraightRedLight, style: Lamp-Lamp1-Red
    Rectangle (699,1110 312x34), "North/South Straight: %d", text variable: Glbl.state1Counter
    Rectangle (699,1144 312x34), "East/West Straight: %d", text variable: Glbl.state2Counter
    Rectangle (699,1178 312x34), "North/South Left: %d", text variable: Glbl.state3Counter
    Rectangle (699,1212 312x34), "East/West Left: %d", text variable: Glbl.state4Counter
    Rectangle (699,1246 312x34), "North Straight/Left: %d", text variable: Glbl.state5Counter
    Rectangle (699,1280 312x34), "South Straight/Left: %d", text variable: Glbl.state6Counter
    Rectangle (699,1314 312x34), "East Straight/Left: %d", text variable: Glbl.state7Counter
    Rectangle (699,1348 312x34), "West Straight/Left: %d", text variable: Glbl.state8Counter
    Rectangle (1433,533 263x110), "ERROR", invisible if: NOT Glbl.error
    Rectangle (1433,643 263x62), "Message: %s", text variable: Glbl.errorMsg
END_VISUALIZATION
